TYPE ST_ItemPK3_OUT2 :
STRUCT
	Identity		:ST_Identity_PK3_OUT2;
	ItemState		:STRING;
	RejectReason	:ST_RejectReason_PK3_OUT2;
	logs			:ST_logs_PK3_OUT2;
	NoRead			:STRING;
END_STRUCT
END_TYPE

(* stored: Version 1.1.0.1, ProductVersion 3.1.4024.13
   DUT ST_ItemPK3_OUT2: Id {aad05c67-7466-4836-bc01-b7f559260bff} *)
